TYPE DUT_UpdateSettingRepositoryByName:
STRUCT  
	return_value	: DINT;
	Name			: STRING(50);
	JsonValue		: STRING(DB.MAX_STRING_SIZE);
END_STRUCT
END_TYPE

(* stored: Version 1.1.0.1, ProductVersion 3.1.4024.15
   DUT DUT_UpdateSettingRepositoryByName: Id {71a508fc-b9c3-41ca-ad9e-213ee6588ec8} *)
